TYPE T_LongSTRING : STRING(1023);
END_TYPE

(* stored: Version 1.1.0.1
   DUT T_LongSTRING: Id {103d09de-a8f7-449e-abe3-62729fec1fa2} *)
